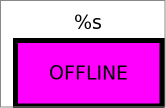
VISUALIZATION Obj_Leak_Detection  // 166x108
VAR_INPUT
	sIndex : STRING;
	bAlarm : BOOL;
	bFault : BOOL;
	bOffline : BOOL;
END_VAR
    Rectangle (13,38 151x70), "%s", colour toggle: bAlarm, text list: 'PDU_Surge_Status', text index: bAlarm
    Rectangle (13,38 151x70), "FAULT", invisible if: not bFault
    Rectangle (10,4 156x37), "%s", text variable: sIndex
    Rectangle (13,38 151x70), "OFFLINE", invisible if: not bOffline
END_VISUALIZATION

(* stored: Version 1.1.0.1, ProductVersion 3.1.4024.12
   Visu Obj_Leak_Detection: Id {0f1f577e-63e3-4794-bb39-f6033a7c3aea} *)
